// TIA Portal V15 export
// export: Created 2018-05-29T12:25:38.1552518Z, ExportSetting WithDefaults, DisplayName Totally Integrated Automation Portal, DisplayVersion V15, DisplayName STEP 7 Professional, DisplayVersion V15, DisplayName WinCC Professional, DisplayVersion V15, DisplayName TIA Portal Openness, DisplayVersion V15
FUNCTION "LT004_fc" : Void   // FC1, STL
TITLE = LT004_fc
{ S7_Optimized_Access := 'TRUE' }
VERSION : 0.1
// test
// stored: AutoNumber true, UDAEnableTagReadback false
BEGIN

NETWORK
TITLE = Main
// comment: PLC1


// Call the CM FB with the corresponding DB instance
      CALL  "BST_ANALOG_400", "LT004"
      ( wVal     := ,
        QfVal    := ,
        LIM_Qb01 := ,
        LIM_Qb02 := ,
        LIM_Qb03 := ,
        LIM_b04  := ,
        QERR     := 
      );
END_FUNCTION
